       //ERROR CAMM SELECTION OR CAM STANDSTILL SELECTION
       ELSIF #statErrorCamSelection OR #statErrorCamStandStillSelection
       THEN
           REGION ----- statErrorCamSelection -----
               // Diagnostic in string
               #status := "LAxisCtrlApcFr_Word2String_Status"(wordStatus := "ERR_LAXISCTRLAPCFR_CAM_SELECTION");
               #errorMC := "LAxisCtrlApcFr_Word2String_Status"(wordStatus := "ERR_LAXISCTRLAPCFR_CAMMANAGEMENT_CAM_NUMBER_SELECTION");
               #errorID := "LAxisCtrlApcFr_Word2String_Status"(wordStatus := "STATUS_FINISHED_NOERROR");
               // Diagnostic in word
               #statDiagnostic.status := "ERR_LAXISCTRLAPCFR_CAM_SELECTION";
               #statDiagnostic.errorMC := "ERR_LAXISCTRLAPCFR_CAMMANAGEMENT_CAM_NUMBER_SELECTION";
               #statDiagnostic.errorID := "STATUS_FINISHED_NOERROR";

               #error := TRUE;
               #statFirstError := TRUE;
           END_REGION

       // ERROR CAMIN
       ELSIF #statCam = 0 AND #statCamIn THEN
           REGION ----- Error Cam Empty -----
               // Diagnostic in string
               #status := "LAxisCtrlApcFr_Word2String_Status"(wordStatus := "ERR_LAXISCTRLAPCFR_CAM_EMPTY");
               #errorMC := "LAxisCtrlApcFr_Word2String_Status"(wordStatus := "ERR_LAXISCTRLAPCFR_CAMMANAGEMENT_CAM_EMPTY");
               #errorID := "LAxisCtrlApcFr_Word2String_Status"(wordStatus := "STATUS_FINISHED_NOERROR");
               // Diagnostic in word
               #statDiagnostic.status := "ERR_LAXISCTRLAPCFR_CAM_EMPTY";
               #statDiagnostic.errorMC := "ERR_LAXISCTRLAPCFR_CAMMANAGEMENT_CAM_EMPTY";
               #statDiagnostic.errorID := "STATUS_FINISHED_NOERROR";

               #error := TRUE;
               #statFirstError := TRUE;
           END_REGION

       // ERROR INTERPOLATE CAM
       ELSIF #statErrorInterpolateCam THEN
           REGION ----- ErrorInterpolateCam -----
               // Diagnostic in string
               #status := "LAxisCtrlApcFr_Word2String_Status"(wordStatus := "ERR_LAXISCTRLAPCFR_INTERPOLATE_CAM");
               #errorMC := "LAxisCtrlApcFr_Word2String_Status"(wordStatus := "ERR_LAXISCTRLAPCFR_CAMMANAGEMENT_INTERPOLATE_CAM");
               #errorID := "LAxisCtrlApcFr_Word2String_ErrorID"(wordErrorID := #instLaxisCtrlApcFr_UnpubMC_Interpolate.instMC.ErrorId, language := #dataAxisConfig.textLanguage);
               // Diagnostic in word
               #statDiagnostic.status := "ERR_LAXISCTRLAPCFR_INTERPOLATE_CAM";
               #statDiagnostic.errorMC := "ERR_LAXISCTRLAPCFR_CAMMANAGEMENT_INTERPOLATE_CAM";
               #statDiagnostic.errorID := #instLaxisCtrlApcFr_UnpubMC_Interpolate.instMC.ErrorId;

               #error := TRUE;
               #statFirstError := TRUE;
           END_REGION

       //ERROR CAMIN CHANGE ON THE FLY
       ELSIF #statErrorCamIChangeOnTheFly THEN
           REGION ----- ErrorChangeCamOnFly -----
               // Diagnostic in string
               #status := "LAxisCtrlApcFr_Word2String_Status"(wordStatus := "ERR_LAXISCTRLAPCFR_CHANGECAMONFLY");
               #errorMC := "LAxisCtrlApcFr_Word2String_Status"(wordStatus := #instLaxisCtrlApcFr_CamInChangeOnTheFly.status);
               #errorID := "LAxisCtrlApcFr_Word2String_ErrorID"(wordErrorID := #instLaxisCtrlApcFr_CamInChangeOnTheFly.subStatus, language := #dataAxisConfig.textLanguage);
               // Diagnostic in word
               #statDiagnostic.status := "ERR_LAXISCTRLAPCFR_CHANGECAMONFLY";
               #statDiagnostic.errorMC := "ERR_LAXISCTRLAPCFR_CAMMANAGEMENT_CHANGECAMONFLY";
               #statDiagnostic.errorID := "ERR_LAXISCTRLAPCFR_CAMMANAGEMENT_NO_CAM_ACTIVE";

               #error := TRUE;
               #statFirstError := TRUE;
           END_REGION

       // ERROR CAMIN STANDSTILL
       ELSIF #statErrorCamInStandStill THEN
           REGION ----- ErrorCamInStandStill -----
               // Diagnostic in string
               #status := "LAxisCtrlApcFr_Word2String_Status"(wordStatus := "ERR_LAXISCTRLAPCFR_CAMINSTANDSTILL");
               #errorMC :="LAxisCtrlApcFr_Word2String_Status"(wordStatus:=#instLAxisCtrlApcFr_CamInStandStill.status);
               #errorID := "LAxisCtrlApcFr_Word2String_ErrorID"(wordErrorID:=#instLAxisCtrlApcFr_CamInStandStill.errorId, language:=#dataAxisConfig.textLanguage);
               // Diagnostic in word
               #statDiagnostic.status := "ERR_LAXISCTRLAPCFR_CAMINSTANDSTILL";
               #statDiagnostic.errorMC := #instLAxisCtrlApcFr_CamInStandStill.status;
               #statDiagnostic.errorID := #instLAxisCtrlApcFr_CamInStandStill.errorId;

               #error := TRUE;
               #statFirstError := TRUE;
           END_REGION

       END_IF;

   END_IF;

   IF #resetAxis THEN
       #error := FALSE;
       #statFirstError := FALSE;

       // Diagnostic in string
       #status := 'STATUS_CALL_FB';
       #errorMC := 'No errorMC';
       #errorID := 'No errorID';
       // Diagnostic in word
       #statDiagnostic.status := "STATUS_FINISHED_NOERROR";
       #statDiagnostic.errorMC := "STATUS_FINISHED_NOERROR";
       #statDiagnostic.errorID := "STATUS_FINISHED_NOERROR";

   END_IF;
   //----------------------------------------------------------------------------------------------
END_REGION
END_FUNCTION_BLOCK
